TYPE (* Value of auxiliary inputs Struct *)
  (* Version 1.0, 2025-07-21, franz *)
  AuxiliaryState_S : STRUCT
    value : USINT := 255;
  END_STRUCT;
END_TYPE
